(* PLC project Tc2_Utilities.FB_SystemTimeToTzSpecificLocalTime Demo, tc3-libraries-kb TwinCAT 3.1 *)
(* stored: creationDateTime 2026-05-11T00:00:00, modificationDateTime 2026-05-11T00:00:00 *)

PROGRAM P_Demo_FB_SystemTimeToTzSpecificLocalTime
  VAR
    fbFB_SystemTimeToTzSpecificLocalTime : FB_SystemTimeToTzSpecificLocalTime;  (* FB_SystemTimeToTzSpecificLocalTime 实例 *)
    bConvert : BOOL := FALSE;
    stTz : TIME_ZONE_INFORMATION;
    stUtc : TIMESTRUCT;
    stLocalTime : TIMESTRUCT;
  END_VAR

// =============================================================================
// 场景：UTC 时间转本地时间。
// 价值：跨版本稳定。
// 验证：给 stUtc 填一个具体 UTC 时间（如 2026-05-11 12:00:00 UTC），触发后 stLocalTime 应为按时区偏移后的值。
// 验证步骤：
//   1. 右键 PLC 项目 → Import PLCopenXML → 选本文件
//   2. 引用 Tc2_Utilities（References → Add library）
//   3. 编译 → 登录 → 运行；按上方『验证』行的指示在线写值观察
// =============================================================================

fbFB_SystemTimeToTzSpecificLocalTime(
    tzInfo := stTz, bExecute := bConvert, stUTC := stUtc,
    stLocal => stLocalTime
);
END_PROGRAM
